FUNCTION_BLOCK FB_CleaningProcessStateCapping EXTENDS FB_CleaningProcessStateBase
VAR_INPUT
END_VAR

VAR_OUTPUT
END_VAR

VAR
END_VAR

METHOD mCleaningOp : BOOL
VAR_INPUT
	sI_Operation : EN_CLEANING_OP;
END_VAR
//Set mode and start process when successful
(*HOA TEST
IF NOT bL_DevOpActive THEN
  bL_DevOpActive := I_ParentCallback.mSetMode(sI_Operation);
  mCleaningOp    := TRUE; //report success
END_IF*) mCleaningOp    := TRUE;

//Switch to production mode if no operation active
IF I_MachineStatus.pSafetyOk AND I_MachineStatus.pMachineReady AND NOT bL_DevOpActive THEN
  IF sI_Operation = eOPCAPENTER THEN
    I_ParentCallback.mChangeState(EN_Cleaning_State.Capping);
  ELSIF sI_Operation = eOPCAPEXIT THEN
    I_ParentCallback.mChangeState(EN_Cleaning_State.CappingExit);
  ELSIF sI_Operation = eOPCLEAN THEN
    I_ParentCallback.mChangeState(EN_Cleaning_State.Cleaning);
  ELSIF sI_Operation = eOPPURGE THEN
    I_ParentCallback.mChangeState(EN_Cleaning_State.Capping);
  END_IF
END_IF
END_METHOD

METHOD mEntryAction
VAR_INPUT
END_VAR
iL_CurrentStep := 0;

// Launch initial command to bring system to service mode
bL_DevOpActive := I_ParentCallback.mSetMode(EN_CLEANING_OP.eOPCAPENTER);
END_METHOD

METHOD mProduction : BOOL
VAR_INPUT
END_VAR
//Switch to production mode if no operation active
IF I_MachineStatus.pSafetyOk AND I_MachineStatus.pMachineReady AND NOT bL_DevOpActive THEN
	I_ParentCallback.mChangeState(EN_Cleaning_State.Production);
END_IF
END_METHOD

METHOD mService : BOOL
VAR_INPUT
END_VAR
//Switch to service mode
IF NOT bL_DevOpActive THEN
	I_ParentCallback.mChangeState(EN_Cleaning_State.Service);
END_IF
END_METHOD

METHOD mStateAction
VAR_INPUT
END_VAR

VAR
	sL_DeviceStatus: ST_CLEANING_DEV_STATUS;
END_VAR
sL_DeviceStatus := I_ParentCallback.pDeviceStatus;
SUPER^.pInitDone := TRUE;

IF bL_DevOpActive THEN
	mDevOp();	
END_IF



//If error go to error mode
IF sL_DeviceStatus.bError THEN
	I_ParentCallback.mChangeState(EN_Cleaning_State.Error);
END_IF
END_METHOD

END_FUNCTION_BLOCK

(* stored: Version 1.1.0.1, ProductVersion 3.1.4024.11
   POU FB_CleaningProcessStateCapping: Id {b1c7a957-1ecc-405b-9047-1f4d47f4aa95}, SpecialFunc None
   Method mCleaningOp: Id {1a8b8234-c65c-4a00-af3f-a93f27b760cf}
   Method mEntryAction: Id {4fab34a5-0860-4616-acf3-576f6c192b00}
   Method mProduction: Id {a588dd05-cdfe-483e-8b5f-f6fa718f556b}
   Method mService: Id {592a7ac9-a875-48a7-9227-28a65bd9f269}
   Method mStateAction: Id {b1d1e10d-9fa1-4eb4-96c9-65ff555e55a4} *)
